// TwinCAT 3 PLC project Untitled1
// ProgramVersion: 3.1.4023.0
// libraries:
//   Tc2_Standard, * (Beckhoff Automation GmbH)
//   Tc2_System, * (Beckhoff Automation GmbH)
//   Tc3_Module, * (Beckhoff Automation GmbH)
// project tree:
//   / PlcTask.TcTTO
//   POUs/ MAIN.TcPOU
// real-time tasks:
//   TASK PlcTask: cycle T#10ms, priority 20, ADS port 350

CONFIGURATION Untitled1
    RESOURCE PLC ON TwinCAT3
        TASK PlcTask(INTERVAL := T#10ms, PRIORITY := 20);
        PROGRAM MAIN WITH PlcTask : MAIN;
    END_RESOURCE
END_CONFIGURATION

// ---- POUs/MAIN.TcPOU
PROGRAM MAIN
VAR
	fileOpen : FB_FileOpen;
	fileWrite : FB_FileWrite;
	fileClose : FB_FileClose;
	step : DINT := 0;
	handle : UINT;
	buffer : ARRAY[1..10] OF BYTE := [65, 66, 67, 13, 10];
	busy : BOOL;
	error : BOOL;
END_VAR

// write to a file as a simple test
CASE step OF
	0:
		fileOpen(
			sNetId:= '', 
			sPathName:= 'C:\TwinCAT\test.txt', 
			nMode:= FOPEN_MODEWRITE, 
			ePath:= PATH_GENERIC, 
			bExecute:= TRUE, 
			tTimeout:= T#5S, 
			bBusy=> busy, 
			bError=> error, 
			nErrId=> , 
			hFile=> handle);
			
			IF NOT fileOpen.bBusy THEN
				step := step + 1;
			END_IF
			
	1:
			fileOpen(bExecute := FALSE);
			step := step + 1;
	2:
		fileWrite(
			sNetId:= '', 
			hFile:= handle, 
			pWriteBuff:= ADR(buffer), 
			cbWriteLen:= 6, 
			bExecute:= TRUE, 
			tTimeout:= T#5S, 
			bBusy=> busy, 
			bError=> error, 
			nErrId=> , 
			cbWrite=> );
		IF NOT fileWrite.bBusy THEN
			step := step + 1;
		END_IF
	3:
		fileWrite(bExecute := FALSE);
		step := step + 1;
	4:
		fileClose(
			sNetId:= '', 
			hFile:= handle, 
			bExecute:= TRUE, 
			tTimeout:= T#5S, 
			bBusy=> busy, 
			bError=> error, 
			nErrId=> );
		IF NOT fileClose.bBusy THEN
			step := step + 1;
		END_IF
	5:
		fileClose(bExecute := FALSE);
		step := step + 1;
END_CASE

END_PROGRAM
